TYPE ST_ServiceExecuteSubStateRecord :
STRUCT
	Step : UDINT;
	Name : STRING(80);
	// UTC timestamp formatted as YYYYMMDDHHMMSSUUU.
	StartTimestamp : STRING(20);
	// Empty while this occurrence is still active.
	EndTimestamp : STRING(20);
END_STRUCT
END_TYPE

(* stored: Version 1.1.0.1, ProductVersion 3.1.4026.18
   DUT ST_ServiceExecuteSubStateRecord: Id {e81d9967-20df-41d0-80f4-593a2a7dfc56} *)
